PROGRAM P_Demo_FB_JsonSaxWriter_GetDocument
VAR
    fbParser : FB_JsonSaxWriter; // 父 FB 实例
    hrErrorCode : HRESULT;
    vRet : STRING(255); // 返回值监视
    bTrigger : BOOL := FALSE; // 在线置 TRUE 触发一次调用
    bTriggerPrev : BOOL;
END_VAR

// =============================================================================
// 场景：拼装完 DOM 后把整份 JSON 拷成 STRING 推到 MQTT broker。
// 价值：一次调用拿到完整序列化字符串。
// 验证：登录 PLC 在线写 bTrigger := TRUE 触发，monitor 返回值/输出参数。具体步骤见下方注释。
// 验证步骤：
//   1. 右键 PLC 项目下 POUs 文件夹 → Add → Existing Item → 选本 .TcPOU 文件
//   2. 引用 Tc3_JsonXml（References → Add library）
//   3. 编译 → 登录 → 运行；按 verify 注释里给出的在线写值操作
// =============================================================================

// 上升沿触发一次方法调用并观察输出。
IF bTrigger AND NOT bTriggerPrev THEN
    vRet := fbParser.GetDocument(
        hrErrorCode => hrErrorCode
    );
END_IF;
bTriggerPrev := bTrigger;

END_PROGRAM

(* stored: Version 1.1.0.1, ProductVersion 3.1.4024.5
   POU P_Demo_FB_JsonSaxWriter_GetDocument: Id {12853a8b-f4b5-597a-8be2-7739282b8b1e}, SpecialFunc None *)
